PROGRAM MAIN
VAR
END_VAR

END_PROGRAM

(* stored: Version 1.1.0.1
   POU MAIN: Id {7f25197a-8e92-4344-b91d-73eaa266427b} *)
